PROGRAM P_Output
VAR
	Mode : E_Modes;
	ManModes : E_ManuelModes;
END_VAR

CASE G_HMI.nCounter OF
	
	E_Modes.Manuel:
	
		G_Enables.bAuto := FALSE;
		G_Enables.bManual := TRUE;
	
		CASE G_HMI.nManuelMode OF
				
			E_ManuelModes.ManDirect:
			
				G_Output.bEnableValveOne := G_Inputs.bEnableButton AND G_Enables.bEnableOne AND NOT(G_Enables.bErrorOne);
				G_Output.bEnableValveTwo := G_Inputs.bEnableButton AND G_Enables.bEnableTwo AND NOT(G_Enables.bErrorTwo);
				G_Output.nValveOneOutput := LREAL_TO_INT(G_OPC.fJoystickMain * 32767.0);
				G_Output.nValveTwoOutput := LREAL_TO_INT(G_OPC.fJoystickJib * 32767.0);
				G_Enables.bManConst := FALSE;
				G_Enables.bManSpeed := FALSE;
				G_Enables.bManDirect := TRUE;
				
			E_ManuelModes.ManConst:
			
				G_Output.bEnableValveOne := G_Inputs.bEnableButton AND G_Enables.bEnableOne AND NOT(G_Enables.bErrorOne);
				G_Output.bEnableValveTwo := G_Inputs.bEnableButton AND G_Enables.bEnableTwo AND NOT(G_Enables.bErrorTwo);
				G_Output.nValveOneOutput := LREAL_TO_INT(G_Parameters.fConst1 * 32767.0) ;
				G_Output.nValveTwoOutput := LREAL_TO_INT(G_Parameters.fConst2 * 32767.0) ;
				G_Enables.bManDirect := FALSE;
				G_Enables.bManSpeed := FALSE;
				G_Enables.bManConst := TRUE;
				
			E_ManuelModes.ManSpeed:
			
				G_Output.bEnableValveOne := G_Inputs.bEnableButton AND G_Enables.bEnableOne AND NOT(G_Enables.bErrorOne);
				G_Output.bEnableValveTwo := G_Inputs.bEnableButton AND G_Enables.bEnableTwo AND NOT(G_Enables.bErrorTwo);
				G_Output.nValveOneOutput := LREAL_TO_INT(G_OPC.fValveOneSignals.fU * 32767.0) ;
				G_Output.nValveTwoOutput := LREAL_TO_INT(G_OPC.fValveTwoSignals.fU * 32767.0) ;
				G_Enables.bManDirect := FALSE;
				G_Enables.bManConst := FALSE;
				G_Enables.bManSpeed := TRUE;
				
			ELSE
			
				G_Enables.bManConst := FALSE;
				G_Enables.bManSpeed := FALSE;
				G_Enables.bManDirect := FALSE;
				
		END_CASE
		
	E_Modes.Off:
		G_Enables.bEnableOne := FALSE;
		G_Enables.bEnableTwo := FALSE;
		G_Enables.bAuto := FALSE;
		G_Enables.bManual := FALSE;

	E_Modes.Auto:
		
		G_Output.bEnableValveOne := G_Inputs.bEnableButton AND G_Enables.bEnableOne AND NOT(G_Enables.bErrorOne);
		G_Output.bEnableValveTwo := G_Inputs.bEnableButton AND G_Enables.bEnableTwo AND NOT(G_Enables.bErrorTwo);
		G_Output.nValveOneOutput := LREAL_TO_INT(G_OPC.fValveOneSignals.fU * 32767.0) * BOOL_TO_INT(G_Enables.bEnableU);
		G_Output.nValveTwoOutput := LREAL_TO_INT(G_OPC.fValveTwoSignals.fU * 32767.0) * BOOL_TO_INT(G_Enables.bEnableU);
		G_Enables.bManual := FALSE;
		G_Enables.bAuto := TRUE;
		
	ELSE
		G_Enables.bEnableOne := FALSE;
		G_Enables.bEnableTwo := FALSE;
		G_Enables.bAuto := FALSE;
		G_Enables.bManual := FALSE;
END_CASE

END_PROGRAM

(* stored: Version 1.1.0.1
   POU P_Output: Id {ea868c64-71e1-491f-a495-e9db7d8a4d4c}, SpecialFunc None *)
